FUNCTION_BLOCK FB_EquipmentModule1 EXTENDS FB_MachineState IMPLEMENTS I_FaultOwner
VAR
    _subState : E_EquipmentModule1State;
	
	// Cylinder 1
    DoubleActingCylinderExtendSensor : FB_DigitalInputHardware(DebounceOnTime := T#0MS, DebounceOffTime := T#0MS, Invert := FALSE);
    DoubleActingCylinderRetractSensor : FB_DigitalInputHardware(DebounceOnTime := T#0MS, DebounceOffTime := T#0MS, Invert := FALSE);
    DoubleActingCylinderExtendSolenoid : FB_DigitalOutputHardware;
    DoubleActingCylinderRetractSolenoid : FB_DigitalOutputHardware;

    CylinderDoubleActing : FB_DoubleActingCylinder
	(
		iCylExtendedSwitch := DoubleActingCylinderExtendSensor,
		iCylRetractedSwitch := DoubleActingCylinderRetractSensor,
		iCylExtend := DoubleActingCylinderExtendSolenoid,
		iCylRetract := DoubleActingCylinderRetractSolenoid,
		eSensorMode := E_SensorMode.BOTH,
		tExtendTimeout := T#3S,
		tRetractTimeout := T#3S
	);

	// Cylinder 2
	_CylinderSingleActingIsInterlocked : BOOL; // Needed because you cant pass a Method as an interface
		
    SingleActingCylinderExtendSensor : FB_DigitalInputHardware(DebounceOnTime := T#0MS, DebounceOffTime := T#0MS, Invert := FALSE);
    SingleActingCylinderRetractSensor : FB_DigitalInputHardware(DebounceOnTime := T#0MS, DebounceOffTime := T#0MS, Invert := FALSE);
    SingleActingCylinderExtendSolenoid : FB_DigitalOutputHardware;

    CylinderSingleActing : FB_SingleActingCylinder
	(
		iCylExtendedSwitch := SingleActingCylinderExtendSensor,
		iCylRetractedSwitch := SingleActingCylinderRetractSensor,
		iCylExtend := SingleActingCylinderExtendSolenoid,
		eSensorMode := E_SensorMode.BOTH,
		tExtendTimeout := T#3S,
		tRetractTimeout := T#3S
	);
	
	// Cylinder Interfaces (not necessarily needed but makes changes easier) 
    iCylinder : I_Cylinder := CylinderDoubleActing; // Polymorphic reference				
    iCylinder2 : I_Cylinder := CylinderSingleActing; // Polymorphic reference

	// Axes
    fbAxis1 : FB_Axis;
	fbAxis2 : FB_Axis;

	// Faults
    fbFaultCyl1Extend : FB_Fault := (
        bAutoReset := FALSE,
        eSeverity := E_FaultSeverity.CRITICAL,
        nCode := 1001,
        sMessage := 'Cylinder 1 extend timeout'
    );
    fbFaultCyl1Retract : FB_Fault := (
        bAutoReset := FALSE,
        eSeverity := E_FaultSeverity.CRITICAL,
        nCode := 1002,
        sMessage := 'Cylinder 1 retract timeout'
    );
	fbFaultCyl1SensorConflict : FB_Fault := (
        bAutoReset := FALSE,
        eSeverity := E_FaultSeverity.CRITICAL,
        nCode := 1003,
        sMessage := 'Cylinder 1 sensor conflict'
    );
	
    fbFaultCyl2Extend  : FB_Fault := (
        bAutoReset := FALSE,
        eSeverity := E_FaultSeverity.CRITICAL,
        nCode := 1011,
        sMessage := 'Cylinder 2 extend timeout'
    );
    fbFaultCyl2Retract : FB_Fault := (
        bAutoReset := FALSE,
        eSeverity := E_FaultSeverity.CRITICAL,
        nCode := 1012,
        sMessage := 'Cylinder 2 retract timeout'
    );
    fbFaultCyl2SensorConflict : FB_Fault := (
        bAutoReset := FALSE,
        eSeverity := E_FaultSeverity.CRITICAL,
        nCode := 1013,
        sMessage := 'Cylinder 2 sensor conflict'
    );
	
	// Equiplevel Faults
    fbFaultSequenceTimeout : FB_Fault := (
        bAutoReset := FALSE,
        eSeverity := E_FaultSeverity.CRITICAL,
        nCode := 9999,
        sMessage := 'Equipment Module 1 Sequence Timeout'
    );
	
	_ipModuleFaults  : ST_EquipmentModuleFaults;
	
	fbFaultManager : FB_FaultManager;
END_VAR

PROPERTY AxisConveryor : I_Axis
GET
AxisConveryor := fbAxis1;
END_GET
END_PROPERTY

PROPERTY CylDouble : I_Cylinder
GET
CylDouble := CylinderDoubleActing;
END_GET
END_PROPERTY

PROPERTY CylSingle : I_Cylinder
GET
CylSingle := CylinderSingleActing;
END_GET
END_PROPERTY

METHOD ExecuteProduction
CASE _subState OF
    E_EquipmentModule1State.EXTEND_CYL1:
        _state := E_MachineState.RUNNING;  // transition from STARTING to RUNNING
        iCylinder.Extend();
        fbAxis1.MoveAbsolute(fPosition := 100.0, fVelocity := 50.0, fAccel := 10000.0, fDecel := 10000.0);
        _subState := E_EquipmentModule1State.WAIT_CYL1;

    E_EquipmentModule1State.WAIT_CYL1:
        IF iCylinder.IsExtended AND fbAxis1.IsIdle THEN
            _subState := E_EquipmentModule1State.EXTEND_CYL2;
        END_IF

    E_EquipmentModule1State.EXTEND_CYL2:
        iCylinder2.Extend();
        fbAxis1.MoveRelative(fDistance := -100.0, fVelocity := 500.0, fAccel := 1000.0, fDecel := 1000.0);
        _subState := E_EquipmentModule1State.WAIT_CYL2;

    E_EquipmentModule1State.WAIT_CYL2:
        IF iCylinder2.IsExtended AND fbAxis1.IsIdle THEN
            _subState := E_EquipmentModule1State.RETRACT_ALL;
        END_IF

    E_EquipmentModule1State.RETRACT_ALL:
        iCylinder.Retract();
        iCylinder2.Retract();
        IF iCylinder.IsRetracted AND iCylinder2.IsRetracted THEN
            _subState := E_EquipmentModule1State.COMPLETE;
        END_IF

    E_EquipmentModule1State.COMPLETE:
        _subState := E_EquipmentModule1State.EXTEND_CYL1;
        _state    := E_MachineState.IDLE;  // sequence done — back to IDLE
END_CASE
END_METHOD

METHOD ExecuteStop : BOOL
VAR_INPUT
END_VAR
// Command cylinders to retract
//iCylinder.Retract();
//iCylinder2.Retract();

// Hold axis
fbAxis1.Halt();

// Wait for everything to reach safe state
(*
IF iCylinder.IsRetracted AND iCylinder2.IsRetracted AND fbAxis.IsIdle THEN
	_subState := E_Module1State.EXTEND_CYL1;  // reset sequence
	_state    := E_MachineState.IDLE;
END_IF
*)
END_METHOD

PROPERTY FaultManager : POINTER TO FB_FaultManager
GET
FaultManager := ADR(fbFaultManager);
END_GET
END_PROPERTY

//FB_Init is always available implicitly and it is used primarily for initialization.
//The return value is not evaluated. For a specific influence, you can also declare the
//methods explicitly and provide additional code there with the standard initialization
//code. You can evaluate the return value.
METHOD FB_Init: BOOL
VAR_INPUT
    bInitRetains: BOOL; // TRUE: the retain variables are initialized (reset warm / reset cold)
    bInCopyCode: BOOL;  // TRUE: the instance will be copied to the copy code afterward (online change)   
END_VAR
VAR
	stFaults : ST_CylinderFaults;
END_VAR
CylinderSingleActing.SetInterlock(_CylinderSingleActingIsInterlocked);

// Inject faults into cylinders
stFaults.ipFaultExtend := fbFaultCyl1Extend;
stFaults.ipFaultRetract := fbFaultCyl1Retract;
stFaults.ipFaultSensorConflict := fbFaultCyl1SensorConflict;
CylinderDoubleActing.SetFaults(stFaults);

stFaults.ipFaultExtend  := fbFaultCyl2Extend;
stFaults.ipFaultRetract := fbFaultCyl2Retract;
stFaults.ipFaultSensorConflict := 0;
CylinderSingleActing.SetFaults(stFaults);

fbFaultManager.RegisterFault(fbFaultCyl1Extend);
fbFaultManager.RegisterFault(fbFaultCyl1Retract);
fbFaultManager.RegisterFault(fbFaultCyl1SensorConflict);
fbFaultManager.RegisterFault(fbFaultCyl2Extend);
fbFaultManager.RegisterFault(fbFaultCyl2Retract);
fbFaultManager.RegisterFault(fbFaultCyl2SensorConflict);
END_METHOD

METHOD RegisterFaults
VAR_INPUT
	ipManager : I_FaultManager;
END_VAR
ipManager.RegisterFault(fbFaultSequenceTimeout);
END_METHOD

METHOD Reset : BOOL
CylDouble.Reset();
CylSingle.Reset();
AxisConveryor.Reset();
END_METHOD

METHOD Run
// Raise Equipment Level Faults
IF _ipModuleFaults.ipEquipmentFault1 <> 0 THEN
	_ipModuleFaults.ipEquipmentFault1.Raise();
END_IF

iCylinder.Run();
iCylinder2.Run();
fbAxis1.Run();
fbAxis2.Run();

_CylinderSingleActingIsInterlocked := iCylinder.IsRetracted;

// Check faults
fbFaultManager.Run();

CASE _state OF
	E_MachineState.IDLE:
		;
	E_MachineState.RUNNING:
		THIS^.ExecuteProduction();
	E_MachineState.STOPPING:
		THIS^.ExecuteStop();
END_CASE
END_METHOD

END_FUNCTION_BLOCK

(* stored: Version 1.1.0.1, ProductVersion 3.1.4026.18
   POU FB_EquipmentModule1: Id {38d16a8a-62f6-449d-b5b6-b3803c34719b}, SpecialFunc None
   Property AxisConveryor: Id {01db86d5-1fae-4a89-b2e0-6901896ecd40}
   Get Get: Id {a3a5387e-7ed8-4ae2-8b7a-790f8d3e8a3c}
   Property CylDouble: Id {ebce16a7-c811-4784-8b4f-26e76274a8aa}
   Get Get: Id {29de9e16-9d45-4e66-b2fe-978c50a278c1}
   Property CylSingle: Id {63420114-3048-4bef-9458-994938ca4880}
   Get Get: Id {9a492868-34a3-4764-a8c8-e9fc08faae86}
   Method ExecuteProduction: Id {6f4e5514-7149-4de1-b003-c9c66d1b37e5}
   Method ExecuteStop: Id {6ee72c22-fe68-47b7-a45a-79809af84a74}
   Property FaultManager: Id {6eca5901-6177-4156-84c2-7ef27f673a19}
   Get Get: Id {e3e1ddc6-09a4-42c1-8a36-9bf317da1cc4}
   Method FB_Init: Id {0978ec87-5bf8-45f4-81e4-84ed87349449}
   Method RegisterFaults: Id {07b45c95-80f0-4792-af6c-634ae497f631}
   Method Reset: Id {acae461e-3042-4b0d-a6e0-1f950953dddd}
   Method Run: Id {d1ecdcb2-ddb2-46de-bca0-86c2216b9294} *)
